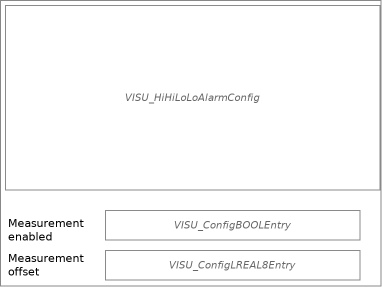
VISUALIZATION VISU_MeasurementConfig  // 382x287
VAR_IN_OUT
	active : MeasurementConfig;
    editable : MeasurementConfig;
END_VAR
    Frame (5,5 375x185)
        shows VISU_HiHiLoLoAlarmConfig(active := active.alarms, editable := editable.alarms)
    Frame (105,210 255x30)
        shows VISU_ConfigBOOLEntry(active := active.enabled, editable := editable.enabled)
    Label (5,210 95x40), "Measurement enabled"
    Label (5,245 95x40), "Measurement offset"
    Frame (105,250 255x30)
        shows VISU_ConfigLREAL8Entry(active := active.offset, editable := editable.offset)
END_VISUALIZATION

(* stored: Version 1.1.0.1, ProductVersion 3.1.4019.2
   Visu VISU_MeasurementConfig: Id {3c45977b-7f91-4362-9229-3b5d6f36b5d7} *)
